(* PLC project Tc2_Utilities.LcomplexAbs Demo, tc3-libraries-kb TwinCAT 3.1 *)
(* stored: creationDateTime 2026-05-12T12:00:00, modificationDateTime 2026-05-12T12:00:00 *)

PROGRAM P_Demo_LcomplexAbs
  VAR
    lcCurrent : LCOMPLEX;
    lrAbs : LREAL;
    bCompute : BOOL;
  END_VAR

            // ============================================================
// Tc2_Utilities.LcomplexAbs 演示程序（FUNCTION，单周期触发）
// ============================================================
// 场景：变频器 d-q 电流幅值 = √(id² + iq²) 用于过电流保护比较。
// 价值：替代手写 `SQRT(re*re + im*im)`；HYPOT 实现在极端值下更稳。
// 验证步骤：
//   1. 把本 PROGRAM 加到 PlcTask 调用列表
//   2. 编译 + 登录
//   3. 在线把 b... 触发位置 TRUE 一个周期
//   4. 观察输出变量是否符合期望
// ============================================================

IF bCompute AND NOT LcomplexIsNaN(lcCurrent) THEN
    // 先判 NaN 避免传播
    lrAbs := LcomplexAbs(lcCurrent);
    bCompute := FALSE;
END_IF;

          
END_PROGRAM
